# EPICS autosave request: iocBoot/ioc13GasLoading/auto_settings.req
file  "Omega_DP41_settings.req",         P=$(P), R=Omega1
file  "Omega_DP41_settings.req",         P=$(P), R=Omega2
file "CARS_motor_settings.req",          P=$(P), M=m1
file "CARS_motor_settings.req",          P=$(P), M=m2
file "CARS_motor_settings.req",          P=$(P), M=m3
file "CARS_motor_settings.req",          P=$(P), M=m4
